FUNCTION LrealBits : ULINT
VAR_INPUT
  x : LREAL;
END_VAR
VAR
  b : POINTER TO ULINT := ADR(x);
END_VAR

LrealBits := b^;

END_FUNCTION

(* stored: Version 1.1.0.1, ProductVersion 3.1.4024.9
   POU LrealBits: Id {2ba3985e-b034-4f38-8371-b63f2efef357}, SpecialFunc None *)
